// TIA Portal V18 export
FUNCTION "Heater" : Void   // FC34, LAD
{ S7_Optimized_Access := 'TRUE' }
VERSION : 0.1
// stored: AutoNumber true, IsIECCheckEnabled false, SetENOAutomatically true, UDAEnableTagReadback false
BEGIN

REGION Network 1 (SCL): Show Heater button if any of the heaters active
   IF "Heater settings"."heater EN 1" OR "Heater settings"."heater EN 2" OR
       "Heater settings"."heater EN 3" OR"Heater settings"."heater EN 4" THEN
       "Heatercontrol"."Show heater Button" := TRUE;
   ELSE
       "Heatercontrol"."Show heater Button" := false;
   END_IF;

   IF "Heatercontrol"."Show heater Button" = false THEN
       "Heatercontrol"."heater ON HMI" := false;
   END_IF;
END_REGION

REGION Network 2 (SCL): Actual temperature of RTD Sensor
   // heaters from 1 to 8 IW144 to IW158 //

   IF "heater1" >= 32767 THEN
       "heater status".temperature.heater1 := 0;
   ELSE
       "heater status".temperature.heater1 := "heater1" / 10;
   END_IF;
   IF "heater2" >= 32767 THEN
       "heater status".temperature.heater2 := 0;
   ELSE
       "heater status".temperature.heater2 := "heater2" / 10;
   END_IF;
   IF "heater3" >= 32767 THEN
       "heater status".temperature.heater3 := 0;
   ELSE
       "heater status".temperature.heater3 := "heater3" / 10;
   END_IF;
   IF "heater4" >= 32767 THEN
       "heater status".temperature.heater4 := 0;
   ELSE
       "heater status".temperature.heater4 := "heater4" / 10;
   END_IF;
END_REGION

REGION Network 3 (SCL): Pt-100 Sensor Connection Okay
   // heaters from 1 to 8 IW144 to IW158 //
   "heater status"."p100 connection okay".heater1 := ("heater1" < 32727);
   "heater status"."p100 connection okay".heater2 := ("heater2" < 32727);
   "heater status"."p100 connection okay".heater3 := ("heater3" < 32727);
   "heater status"."p100 connection okay".heater4 := ("heater4" < 32727);
END_REGION

REGION Network 4 (SCL): alarm
   "Alarm_DB".input.alarm[3] := NOT ("heater status"."p100 connection okay".heater1) AND "Heater settings"."heater EN 1"; //A12-Heater1 sensor fault
   "Alarm_DB".input.alarm[4] := NOT ("heater status"."p100 connection okay".heater2) AND "Heater settings"."heater EN 2";  //A13-Heater1 sensor fault
   "Alarm_DB".input.alarm[5] := NOT ("heater status"."p100 connection okay".heater3) AND "Heater settings"."heater EN 3"; //A14-Heater3 sensor fault
   "Alarm_DB".input.alarm[6] := NOT ("heater status"."p100 connection okay".heater4) AND "Heater settings"."heater EN 4";  //A15-Heater4 sensor fault


   "Alarm_DB".input.alarm[28] := "heater status"."Limit Over temperature".heater1; //"A21- Heater 1overtemperature"
   "Alarm_DB".input.alarm[29] := "heater status"."Limit Over temperature".heater2; //"A22- Heater2 overtemperature"
   "Alarm_DB".input.alarm[30] := "heater status"."Limit Over temperature".heater3; //"A23- Heater3 overtemperature"
   "Alarm_DB".input.alarm[31] := "heater status"."Limit Over temperature".heater4; //"A24- Heater4 overtemperature"

   "Alarm_DB".input.alarm[24] := ("heater status"."Dispensing Stop under temperature heater"[1] AND "Heater settings"."heater EN 1") OR "heater status"."Limit under temperature".heater1;
   "Alarm_DB".input.alarm[25] := ("heater status"."Dispensing Stop under temperature heater"[2] AND "Heater settings"."heater EN 2") OR "heater status"."Limit under temperature".heater2;
   "Alarm_DB".input.alarm[26] := ("heater status"."Dispensing Stop under temperature heater"[3] AND "Heater settings"."heater EN 3") OR "heater status"."Limit under temperature".heater3;
   "Alarm_DB".input.alarm[27] := ("heater status"."Dispensing Stop under temperature heater"[4] AND "Heater settings"."heater EN 4") OR "heater status"."Limit under temperature".heater4;
END_REGION

REGION Network 5: heater 1- Vessel heating sleeve A component
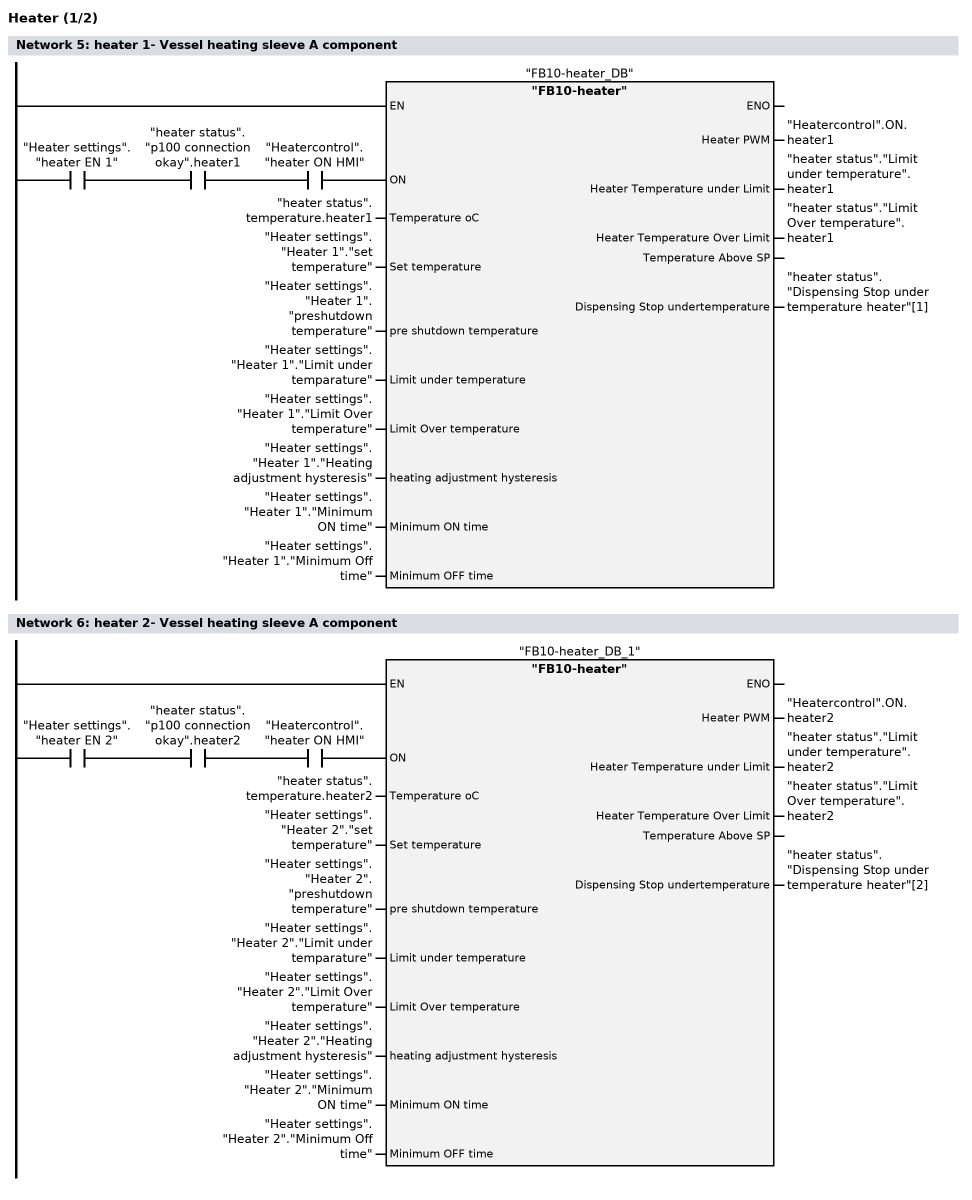
   RUNG wire#powerrail
      "FB10-heater_DB"(ON := wire#w1, "Temperature oC" := "heater status".temperature.heater1, "Set temperature" := "Heater settings"."Heater 1"."set temperature", "pre shutdown temperature" := "Heater settings"."Heater 1"."preshutdown temperature", "Limit under temperature" := "Heater settings"."Heater 1"."Limit under temparature", "Limit Over temperature" := "Heater settings"."Heater 1"."Limit Over temperature", "heating adjustment hysteresis" := "Heater settings"."Heater 1"."Heating adjustment hysteresis", "Minimum ON time" := "Heater settings"."Heater 1"."Minimum ON time", "Minimum OFF time" := "Heater settings"."Heater 1"."Minimum Off time", "Heater PWM" => "Heatercontrol".ON.heater1, "Heater Temperature under Limit" => "heater status"."Limit under temperature".heater1, "Heater Temperature Over Limit" => "heater status"."Limit Over temperature".heater1, "Temperature Above SP" =>, "Dispensing Stop undertemperature" => "heater status"."Dispensing Stop under temperature heater"[1])
   END_RUNG
   RUNG wire#powerrail
      Contact( "Heater settings"."heater EN 1" )
      Contact( "heater status"."p100 connection okay".heater1 )
      Contact( "Heatercontrol"."heater ON HMI" )
   END_RUNG wire#w1
   // the same network as SCL:
   "FB10-heater_DB"(ON := "Heater settings"."heater EN 1" AND "heater status"."p100 connection okay".heater1 AND "Heatercontrol"."heater ON HMI",   // "FB10-heater"
                    "Temperature oC" := "heater status".temperature.heater1,
                    "Set temperature" := "Heater settings"."Heater 1"."set temperature",
                    "pre shutdown temperature" := "Heater settings"."Heater 1"."preshutdown temperature",
                    "Limit under temperature" := "Heater settings"."Heater 1"."Limit under temparature",
                    "Limit Over temperature" := "Heater settings"."Heater 1"."Limit Over temperature",
                    "heating adjustment hysteresis" := "Heater settings"."Heater 1"."Heating adjustment hysteresis",
                    "Minimum ON time" := "Heater settings"."Heater 1"."Minimum ON time",
                    "Minimum OFF time" := "Heater settings"."Heater 1"."Minimum Off time",
                    "Heater PWM" => "Heatercontrol".ON.heater1,
                    "Heater Temperature under Limit" => "heater status"."Limit under temperature".heater1,
                    "Heater Temperature Over Limit" => "heater status"."Limit Over temperature".heater1,
                    "Dispensing Stop undertemperature" => "heater status"."Dispensing Stop under temperature heater"[1]);
END_REGION

REGION Network 6: heater 2- Vessel heating sleeve A component
   RUNG wire#powerrail
      "FB10-heater_DB_1"(ON := wire#w1, "Temperature oC" := "heater status".temperature.heater2, "Set temperature" := "Heater settings"."Heater 2"."set temperature", "pre shutdown temperature" := "Heater settings"."Heater 2"."preshutdown temperature", "Limit under temperature" := "Heater settings"."Heater 2"."Limit under temparature", "Limit Over temperature" := "Heater settings"."Heater 2"."Limit Over temperature", "heating adjustment hysteresis" := "Heater settings"."Heater 2"."Heating adjustment hysteresis", "Minimum ON time" := "Heater settings"."Heater 2"."Minimum ON time", "Minimum OFF time" := "Heater settings"."Heater 2"."Minimum Off time", "Heater PWM" => "Heatercontrol".ON.heater2, "Heater Temperature under Limit" => "heater status"."Limit under temperature".heater2, "Heater Temperature Over Limit" => "heater status"."Limit Over temperature".heater2, "Temperature Above SP" =>, "Dispensing Stop undertemperature" => "heater status"."Dispensing Stop under temperature heater"[2])
   END_RUNG
   RUNG wire#powerrail
      Contact( "Heater settings"."heater EN 2" )
      Contact( "heater status"."p100 connection okay".heater2 )
      Contact( "Heatercontrol"."heater ON HMI" )
   END_RUNG wire#w1
   // the same network as SCL:
   "FB10-heater_DB_1"(ON := "Heater settings"."heater EN 2" AND "heater status"."p100 connection okay".heater2 AND "Heatercontrol"."heater ON HMI",   // "FB10-heater"
                      "Temperature oC" := "heater status".temperature.heater2,
                      "Set temperature" := "Heater settings"."Heater 2"."set temperature",
                      "pre shutdown temperature" := "Heater settings"."Heater 2"."preshutdown temperature",
                      "Limit under temperature" := "Heater settings"."Heater 2"."Limit under temparature",
                      "Limit Over temperature" := "Heater settings"."Heater 2"."Limit Over temperature",
                      "heating adjustment hysteresis" := "Heater settings"."Heater 2"."Heating adjustment hysteresis",
                      "Minimum ON time" := "Heater settings"."Heater 2"."Minimum ON time",
                      "Minimum OFF time" := "Heater settings"."Heater 2"."Minimum Off time",
                      "Heater PWM" => "Heatercontrol".ON.heater2,
                      "Heater Temperature under Limit" => "heater status"."Limit under temperature".heater2,
                      "Heater Temperature Over Limit" => "heater status"."Limit Over temperature".heater2,
                      "Dispensing Stop undertemperature" => "heater status"."Dispensing Stop under temperature heater"[2]);
END_REGION

REGION Network 7: heater 3- Heating sleeve flowmeter A component
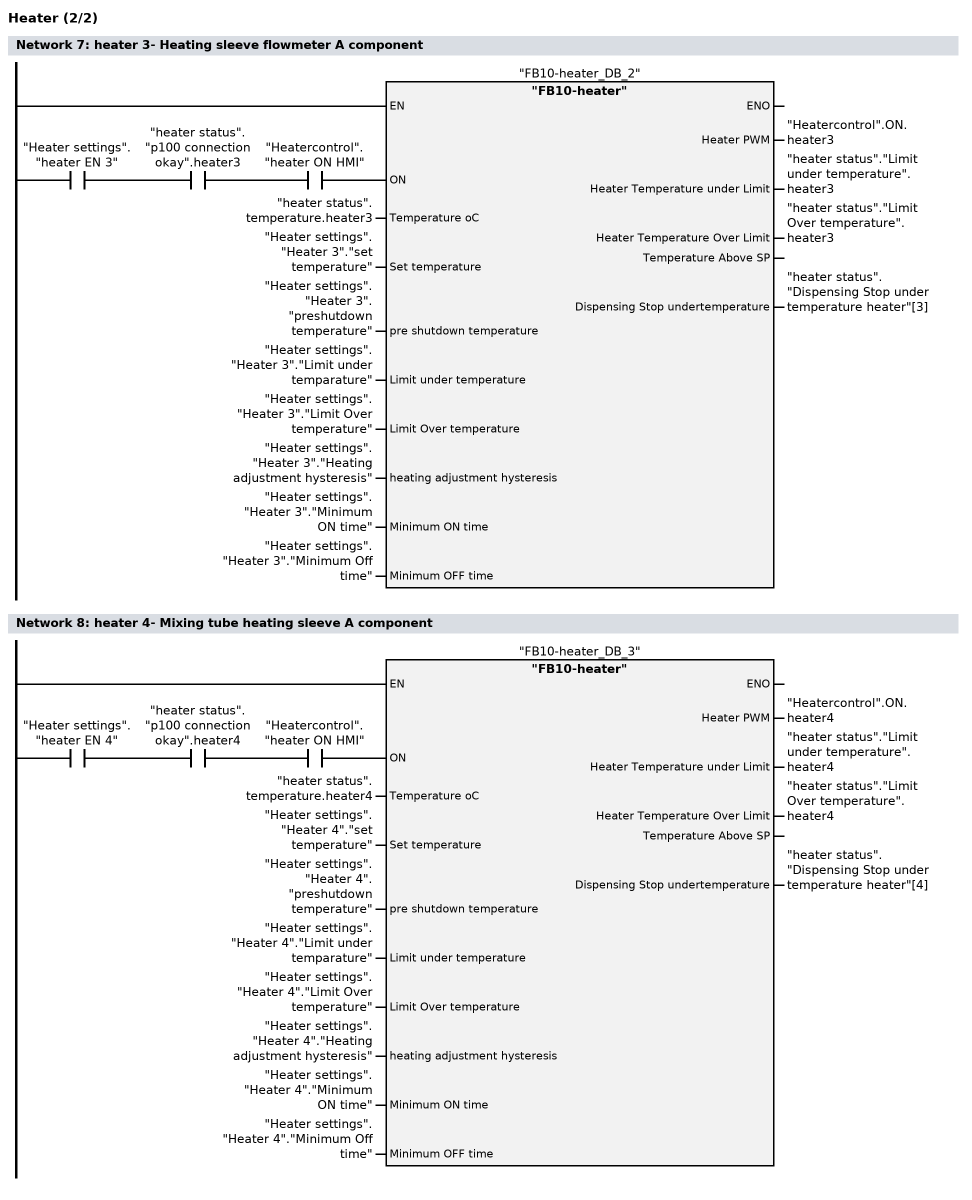
   RUNG wire#powerrail
      "FB10-heater_DB_2"(ON := wire#w1, "Temperature oC" := "heater status".temperature.heater3, "Set temperature" := "Heater settings"."Heater 3"."set temperature", "pre shutdown temperature" := "Heater settings"."Heater 3"."preshutdown temperature", "Limit under temperature" := "Heater settings"."Heater 3"."Limit under temparature", "Limit Over temperature" := "Heater settings"."Heater 3"."Limit Over temperature", "heating adjustment hysteresis" := "Heater settings"."Heater 3"."Heating adjustment hysteresis", "Minimum ON time" := "Heater settings"."Heater 3"."Minimum ON time", "Minimum OFF time" := "Heater settings"."Heater 3"."Minimum Off time", "Heater PWM" => "Heatercontrol".ON.heater3, "Heater Temperature under Limit" => "heater status"."Limit under temperature".heater3, "Heater Temperature Over Limit" => "heater status"."Limit Over temperature".heater3, "Temperature Above SP" =>, "Dispensing Stop undertemperature" => "heater status"."Dispensing Stop under temperature heater"[3])
   END_RUNG
   RUNG wire#powerrail
      Contact( "Heater settings"."heater EN 3" )
      Contact( "heater status"."p100 connection okay".heater3 )
      Contact( "Heatercontrol"."heater ON HMI" )
   END_RUNG wire#w1
   // the same network as SCL:
   "FB10-heater_DB_2"(ON := "Heater settings"."heater EN 3" AND "heater status"."p100 connection okay".heater3 AND "Heatercontrol"."heater ON HMI",   // "FB10-heater"
                      "Temperature oC" := "heater status".temperature.heater3,
                      "Set temperature" := "Heater settings"."Heater 3"."set temperature",
                      "pre shutdown temperature" := "Heater settings"."Heater 3"."preshutdown temperature",
                      "Limit under temperature" := "Heater settings"."Heater 3"."Limit under temparature",
                      "Limit Over temperature" := "Heater settings"."Heater 3"."Limit Over temperature",
                      "heating adjustment hysteresis" := "Heater settings"."Heater 3"."Heating adjustment hysteresis",
                      "Minimum ON time" := "Heater settings"."Heater 3"."Minimum ON time",
                      "Minimum OFF time" := "Heater settings"."Heater 3"."Minimum Off time",
                      "Heater PWM" => "Heatercontrol".ON.heater3,
                      "Heater Temperature under Limit" => "heater status"."Limit under temperature".heater3,
                      "Heater Temperature Over Limit" => "heater status"."Limit Over temperature".heater3,
                      "Dispensing Stop undertemperature" => "heater status"."Dispensing Stop under temperature heater"[3]);
END_REGION

REGION Network 8: heater 4- Mixing tube heating sleeve A component
   RUNG wire#powerrail
      "FB10-heater_DB_3"(ON := wire#w1, "Temperature oC" := "heater status".temperature.heater4, "Set temperature" := "Heater settings"."Heater 4"."set temperature", "pre shutdown temperature" := "Heater settings"."Heater 4"."preshutdown temperature", "Limit under temperature" := "Heater settings"."Heater 4"."Limit under temparature", "Limit Over temperature" := "Heater settings"."Heater 4"."Limit Over temperature", "heating adjustment hysteresis" := "Heater settings"."Heater 4"."Heating adjustment hysteresis", "Minimum ON time" := "Heater settings"."Heater 4"."Minimum ON time", "Minimum OFF time" := "Heater settings"."Heater 4"."Minimum Off time", "Heater PWM" => "Heatercontrol".ON.heater4, "Heater Temperature under Limit" => "heater status"."Limit under temperature".heater4, "Heater Temperature Over Limit" => "heater status"."Limit Over temperature".heater4, "Temperature Above SP" =>, "Dispensing Stop undertemperature" => "heater status"."Dispensing Stop under temperature heater"[4])
   END_RUNG
   RUNG wire#powerrail
      Contact( "Heater settings"."heater EN 4" )
      Contact( "heater status"."p100 connection okay".heater4 )
      Contact( "Heatercontrol"."heater ON HMI" )
   END_RUNG wire#w1
   // the same network as SCL:
   "FB10-heater_DB_3"(ON := "Heater settings"."heater EN 4" AND "heater status"."p100 connection okay".heater4 AND "Heatercontrol"."heater ON HMI",   // "FB10-heater"
                      "Temperature oC" := "heater status".temperature.heater4,
                      "Set temperature" := "Heater settings"."Heater 4"."set temperature",
                      "pre shutdown temperature" := "Heater settings"."Heater 4"."preshutdown temperature",
                      "Limit under temperature" := "Heater settings"."Heater 4"."Limit under temparature",
                      "Limit Over temperature" := "Heater settings"."Heater 4"."Limit Over temperature",
                      "heating adjustment hysteresis" := "Heater settings"."Heater 4"."Heating adjustment hysteresis",
                      "Minimum ON time" := "Heater settings"."Heater 4"."Minimum ON time",
                      "Minimum OFF time" := "Heater settings"."Heater 4"."Minimum Off time",
                      "Heater PWM" => "Heatercontrol".ON.heater4,
                      "Heater Temperature under Limit" => "heater status"."Limit under temperature".heater4,
                      "Heater Temperature Over Limit" => "heater status"."Limit Over temperature".heater4,
                      "Dispensing Stop undertemperature" => "heater status"."Dispensing Stop under temperature heater"[4]);
END_REGION

REGION Network 9 (SCL): Stop Dispensing when Temperature Not Okay During under temperature Without making heater ON
   IF ("heater status"."Dispensing Stop under temperature heater"[1] AND "Heater settings"."heater EN 1") OR
       ("heater status"."Dispensing Stop under temperature heater"[2] AND "Heater settings"."heater EN 2") OR
       ("heater status"."Dispensing Stop under temperature heater"[3] AND "Heater settings"."heater EN 3") OR
       ("heater status"."Dispensing Stop under temperature heater"[4] AND "Heater settings"."heater EN 4")OR
       "heater status".heater_nok
   THEN
     "heater status"."Critical Fault Stop Dispense Temperature NOK" := 1;
   ELSE
     "heater status"."Critical Fault Stop Dispense Temperature NOK" := 0;
   END_IF;
END_REGION
END_FUNCTION
